Yaskawa INFORM job: small_pipe_bent_planes_program.JBI

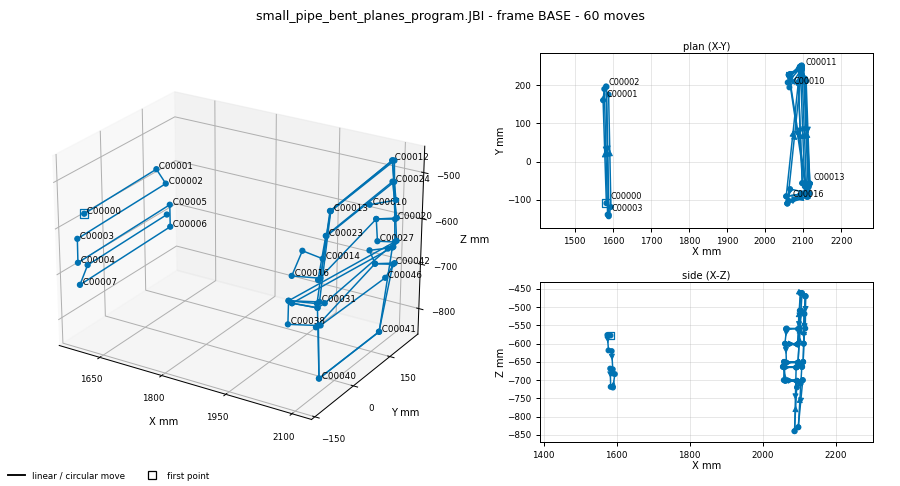
[picture p0: tool path of small_pipe_bent_planes_program.JBI in frame BASE, 60 of 63 moves have a stored position in this frame; points joined in program order, loops and branches not executed]
/JOB
//NAME small_pipe_bent_planes_program
//POS
///NPOS 60,0,60,0,0,0
///TOOL 0
///POSTYPE BASE
///RECTAN
///RCONF 0,0,0,0,0,0,0,0,0,0,0,0,0,0,0,0,0,0,0,0,0,0,0,0
C00000=1583.102048,-109.522293,-578.021566,5.000000,-86.564629,-175.000000
C00001=1574.477575,160.870208,-576.630430,5.000000,-86.564629,-175.000000
C00002=1577.537987,190.525402,-618.908991,5.000000,-86.564629,-175.000000
C00003=1586.345971,-139.488264,-620.710008,5.000000,-86.564629,-175.000000
C00004=1589.278943,-144.016536,-670.657162,5.000000,-86.564629,-175.000000
C00005=1582.275774,197.550532,-668.666239,5.000000,-86.564629,-175.000000
C00006=1583.566574,196.248211,-718.689199,5.000000,-86.564629,-175.000000
C00007=1589.683773,-140.282531,-720.697752,5.000000,-86.564629,-175.000000
C00008=1595.034079,-119.529458,-683.718777,5.000000,-86.564629,-175.000000
C00009=1588.990055,175.969061,-681.995502,180.000000,-60.000000,0.000000
C00010=2063.963227,194.789025,-559.880778,175.000000,-86.807196,5.000000
C00011=2096.978939,244.244403,-560.076331,5.000000,-89.800960,140.186608
C00012=2103.323013,210.351781,-461.887798,175.000000,-57.228100,-29.480841
C00013=2117.850634,-58.096014,-470.119845,175.000000,-61.123555,42.991608
C00014=2116.963551,-83.829209,-558.590747,175.000000,-89.831734,50.186024
C00015=2065.813115,-72.195312,-558.683177,-170.024451,-90.000000,5.000000
C00016=2061.039921,-102.962995,-600.327595,175.000000,-86.807196,5.000000
C00017=2112.710964,-83.336860,-600.383425,175.000000,-89.802724,49.772340
C00018=2116.173213,-57.681346,-470.337439,175.000000,-61.244785,42.683241
C00019=2104.450843,210.724956,-461.499356,-175.000000,-57.036175,-29.746535
C00020=2095.938378,244.868802,-602.137892,5.000000,-89.763198,139.773156
C00021=2063.505114,225.355378,-602.064733,-170.024451,-90.000000,5.000000
C00022=2112.641912,-92.533344,-600.334766,175.000000,-89.802724,49.772340
C00023=2113.409971,-67.113267,-518.568817,175.000000,-61.245084,42.682974
C00024=2101.807969,217.485038,-509.816818,175.000000,-57.036675,-29.745505
C00025=2095.990914,251.865640,-602.174913,5.000000,-89.763198,139.773156
C00026=2063.505114,225.355378,-602.064733,-170.024451,-90.000000,5.000000
C00027=2065.082494,229.912947,-652.253254,175.000000,-86.807196,5.000000
C00028=2096.829172,245.249030,-652.310982,5.000000,-89.734219,139.460410
C00029=2107.996461,210.999483,-461.350721,-175.000000,-56.888511,-29.945850
C00030=2117.595171,-57.361913,-470.648447,-175.000000,-61.334825,42.449056
C00031=2111.171149,-83.049109,-650.352680,175.000000,-89.781030,49.459394
C00032=2058.816123,-110.065193,-650.247267,-170.024451,-90.000000,5.000000
C00033=2096.958135,252.245867,-652.352266,5.000000,-89.734219,139.460410
C00034=2105.432441,217.761326,-509.671179,175.000000,-56.888423,-29.945963
C00035=2114.731202,-66.793745,-518.873939,175.000000,-61.335011,42.448795
C00036=2111.001642,-92.245593,-650.298417,175.000000,-89.781030,49.459394
C00037=2058.816123,-110.065193,-650.247267,-170.024451,-90.000000,5.000000
C00038=2057.983146,-110.298882,-700.277988,175.000000,-86.807196,5.000000
C00039=2109.962964,-83.607319,-700.375403,175.000000,-89.793856,49.644794
C00040=2097.673747,-56.661640,-829.419276,-5.000000,-62.681911,-139.445962
C00041=2087.295624,205.815567,-840.222710,5.000000,-58.221339,152.429846
C00042=2094.180916,244.636805,-702.212899,5.000000,-89.751430,139.645688
C00043=2062.027038,227.815804,-702.150919,-170.024451,-90.000000,5.000000
C00044=2109.852973,-92.803803,-700.324460,175.000000,-89.793856,49.644794
C00045=2104.262736,-65.273424,-709.269233,5.000000,-62.682003,-139.445983
C00046=2094.077271,213.397011,-720.161930,-5.000000,-58.221624,152.430250
C00047=2094.264599,251.633643,-702.251657,5.000000,-89.751430,139.645688
C00048=2062.027038,227.815804,-702.150919,-170.024451,-90.000000,5.000000
C00049=2059.440700,207.711864,-665.384481,175.000000,-86.807196,5.000000
C00050=2091.793514,244.451792,-665.558638,-5.000000,-89.748727,139.616493
C00051=2087.679044,205.837409,-840.277210,5.000000,-58.205559,152.413665
C00052=2097.862457,-56.634543,-829.407375,-5.000000,-62.692511,-139.465973
C00053=2107.348664,-83.800993,-663.702115,175.000000,-89.791830,49.615580
C00054=2055.557679,-91.446831,-663.710324,-170.024451,-90.000000,5.000000
C00055=2091.848704,248.703766,-665.582433,5.000000,-89.748727,139.616493
C00056=2097.870568,214.173934,-654.858064,175.000000,-56.961777,-29.847004
C00057=2108.477281,-57.986553,-663.907766,175.000000,-61.290564,42.565729
C00058=2107.354863,-83.323409,-663.704787,-175.000000,-89.791830,49.615580
C00059=2055.557679,-91.446831,-663.710324,180.000000,-60.000000,0.000000
///POSTYPE PULSE
///PULSE
EC00000=13312.0
EC00001=13312.0
EC00002=13312.0
EC00003=13312.0
EC00004=13312.0
EC00005=13312.0
EC00006=13312.0
EC00007=13312.0
EC00008=13312.0
EC00009=13312.0
EC00010=194560.0
EC00011=194560.0
EC00012=194560.0
EC00013=194560.0
EC00014=194560.0
EC00015=194560.0
EC00016=194560.0
EC00017=194560.0
EC00018=194560.0
EC00019=194560.0
EC00020=194560.0
EC00021=194560.0
EC00022=194560.0
EC00023=194560.0
EC00024=194560.0
EC00025=194560.0
EC00026=194560.0
EC00027=194560.0
EC00028=194560.0
EC00029=194560.0
EC00030=194560.0
EC00031=194560.0
EC00032=194560.0
EC00033=194560.0
EC00034=194560.0
EC00035=194560.0
EC00036=194560.0
EC00037=194560.0
EC00038=194560.0
EC00039=194560.0
EC00040=194560.0
EC00041=194560.0
EC00042=194560.0
EC00043=194560.0
EC00044=194560.0
EC00045=194560.0
EC00046=194560.0
EC00047=194560.0
EC00048=194560.0
EC00049=194560.0
EC00050=194560.0
EC00051=194560.0
EC00052=194560.0
EC00053=194560.0
EC00054=194560.0
EC00055=194560.0
EC00056=194560.0
EC00057=194560.0
EC00058=194560.0
EC00059=194560.0
//INST
///DATE 2023/08/16 14:34
///ATTR SC,RW,RJ
////FRAME BASE
///GROUP1 RB1,ST1
NOP
MOVJ P009 EX000 VJ=15.00
MOVJ C00000 EC00000 VJ=15.0
CALL JOB:SPYON
MOVL C00001 EC00001 V=150.0
MOVL C00002 EC00002 V=150.0
MOVL C00003 EC00003 V=150.0
MOVL C00004 EC00004 V=150.0
MOVL C00005 EC00005 V=150.0
MOVL C00006 EC00006 V=150.0
MOVL C00007 EC00007 V=150.0
MOVL C00008 EC00008 V=150.0
MOVL C00009 EC00009 V=150.0
CALL JOB:SPYOF
MOVJ P009 VJ=15.00
MOVJ C00010 EC00010 VJ=15.0
CALL JOB:SPYON
MOVL C00011 EC00011 V=150.0
MOVL C00012 EC00012 V=150.0
MOVL C00013 EC00013 V=150.0
MOVL C00014 EC00014 V=150.0
MOVL C00015 EC00015 V=150.0
MOVL C00016 EC00016 V=150.0
MOVL C00017 EC00017 V=150.0
MOVL C00018 EC00018 V=150.0
MOVL C00019 EC00019 V=150.0
MOVL C00020 EC00020 V=150.0
MOVL C00021 EC00021 V=150.0
MOVL C00022 EC00022 V=150.0
MOVL C00023 EC00023 V=150.0
MOVL C00024 EC00024 V=150.0
MOVL C00025 EC00025 V=150.0
MOVL C00026 EC00026 V=150.0
MOVL C00027 EC00027 V=150.0
MOVL C00028 EC00028 V=150.0
MOVL C00029 EC00029 V=150.0
MOVL C00030 EC00030 V=150.0
MOVL C00031 EC00031 V=150.0
MOVL C00032 EC00032 V=150.0
MOVL C00033 EC00033 V=150.0
MOVL C00034 EC00034 V=150.0
MOVL C00035 EC00035 V=150.0
MOVL C00036 EC00036 V=150.0
MOVL C00037 EC00037 V=150.0
MOVL C00038 EC00038 V=150.0
MOVL C00039 EC00039 V=150.0
MOVL C00040 EC00040 V=150.0
MOVL C00041 EC00041 V=150.0
MOVL C00042 EC00042 V=150.0
MOVL C00043 EC00043 V=150.0
MOVL C00044 EC00044 V=150.0
MOVL C00045 EC00045 V=150.0
MOVL C00046 EC00046 V=150.0
MOVL C00047 EC00047 V=150.0
MOVL C00048 EC00048 V=150.0
MOVL C00049 EC00049 V=150.0
MOVL C00050 EC00050 V=150.0
MOVL C00051 EC00051 V=150.0
MOVL C00052 EC00052 V=150.0
MOVL C00053 EC00053 V=150.0
MOVL C00054 EC00054 V=150.0
MOVL C00055 EC00055 V=150.0
MOVL C00056 EC00056 V=150.0
MOVL C00057 EC00057 V=150.0
MOVL C00058 EC00058 V=150.0
MOVL C00059 EC00059 V=150.0
CALL JOB:SPYOF
MOVJ P009 VJ=15.00
END
